{attribute 'qualified_only'}
{attribute 'strict'}
{attribute 'to_string'}
TYPE eSeverity :
(
	Info := 0,
	Warning := 1,
	Error := 2,
	Critical := 3
);
END_TYPE

(* stored: Version 1.1.0.1, ProductVersion 3.1.4026.18
   DUT eSeverity: Id {a1b2c3d4-2222-2222-2222-222222222222} *)
